Fanuc TP program (LS listing): MON_T1.LS

/PROG  MON_T1	  Cond
/ATTR
OWNER		= MNEDITOR;
COMMENT		= "MONITOR TOOL 1";
PROG_SIZE	= 231;
CREATE		= DATE 17-03-16  TIME 14:00:18;
MODIFIED	= DATE 17-03-16  TIME 14:33:38;
FILE_NAME	= MON_PRES;
VERSION		= 0;
LINE_COUNT	= 1;
MEMORY_SIZE	= 607;
PROTECT		= READ_WRITE;
TCD:  STACK_SIZE	= 0,
      TASK_PRIORITY	= 50,
      TIME_SLICE	= 0,
      BUSY_LAMP_OFF	= 0,
      ABORT_REQUEST	= 0,
      PAUSE_REQUEST	= 0;
DEFAULT_GROUP	= *,*,*,*,*;
CONTROL_CODE	= 00000000 00000000;
/APPL

AUTO_SINGULARITY_HEADER;
  ENABLE_SINGULARITY_AVOIDANCE   : TRUE;
/MN
   1:  WHEN RI[R[106]]=ON,CALL MON_T1ALM ;
/POS
/END
